{attribute 'qualified_only'}
{attribute 'strict'}
TYPE E_SystemMode :
(
    MANUAL := 0,         // 수동 모드
    AUTO := 1,           // 자동 모드
    ALARM := 2           // 알람 모드
) := MANUAL;
END_TYPE

(* stored: Version 1.1.0.1
   DUT E_SystemMode: Id {12345678-1234-1234-1234-123456789010} *)
